FUNCTION_BLOCK FB_BaseMotor

VAR
	mcAxis: 			AXIS_REF;
	eSMState:			E_MoveState;
	
	mcPower: 			MC_Power;
	mcPower_Outputs:	ST_McOutputs;
	
	mcReset: 			MC_Reset;
	mcReset_Outputs:	ST_McOutputs;
	
	mcStop:				MC_Stop;
	mcStop_Outputs:		ST_McOutputs;
	
	mcMoveAbs1: 			MC_MoveAbsolute;
	mcMoveAbs1_Outputs: 	ST_McOutputs;

	mcMoveAbs2: 			MC_MoveAbsolute;
	mcMoveAbs2_Outputs: 	ST_McOutputs;
	
	mcHome:				MC_Home;
	mcHome_Outputs:		ST_McOutputs;
	
END_VAR

(* update the axis status at the beginning of each cycle *)
mcAxis();

(* move axis using a state machine *)
CASE eSMState OF

	MOVESTATE_INIT :	(* initialisation *)
		(* initialize all function blocks *)
		mcMoveAbs1.Execute := FALSE;
		mcReset.Execute := FALSE;
		eSMState := MOVESTATE_ENABLE;

	MOVESTATE_ENABLE :
		mcPower.Enable := TRUE;
		mcPower.Enable_Positive := TRUE;
		mcPower.Enable_Negative := TRUE;
		IF mcPower.Status THEN
			eSMState := MOVESTATE_FORWARD;
		ELSIF mcPower.Error THEN
			eSMState := MOVESTATE_ERROR;
		END_IF

	MOVESTATE_FORWARD :							(* start to first position *)
		mcMoveAbs1.Position := 1500;				(* start to intermediate tartet position *)
		mcMoveAbs1.Velocity := 500;				(* medium velocity level *)
		mcMoveAbs1.BufferMode := MC_Buffered;
		mcMoveAbs1.Execute := TRUE;
		IF mcMoveAbs1.Active  THEN
			(* axis is executing job but is not yet finished *)
			mcMoveAbs1.Execute := FALSE;
			(* leave this state and buffer a second command *)
			eSMState := MOVESTATE_NEWTARGETPOSITION;
		ELSIF mcMoveAbs1.CommandAborted OR mcMoveAbs1.Error THEN
			eSMState := MOVESTATE_ERROR;
		END_IF

	MOVESTATE_NEWTARGETPOSITION :						(* change target position while moving *)
		(* start a buffered motion command while axis is moving *)
		mcMoveAbs2.Position := 5000;						(* start to final target *)
		mcMoveAbs2.Velocity := 1500;						(* increase velocity *)
		mcMoveAbs2.BufferMode := MC_BlendingPrevious; 		(* use velocity of previous command till intermediate target position position *)
		mcMoveAbs2.Execute := TRUE;
		IF mcMoveAbs2.Done THEN
			mcMoveAbs2.Execute := FALSE;
			eSMState := MOVESTATE_BACKWARDS;
		ELSIF mcMoveAbs2.CommandAborted OR mcMoveAbs2.Error THEN
			eSMState := MOVESTATE_ERROR;
		END_IF

	MOVESTATE_BACKWARDS :							(* move back to initial position *)
		mcMoveAbs1.Position := 100;					(* position close to initial position *)
		mcMoveAbs1.Velocity := 2000;				(* high velocity *)
		mcMoveAbs1.BufferMode := MC_Buffered;
		mcMoveAbs1.Execute := TRUE;
		IF mcMoveAbs1.Active THEN
			(* axis is executing job but is not yet finished *)
			mcMoveAbs1.Execute := FALSE;
			(* leave this state and buffer a second command *)
			eSMState := MOVESTATE_BACKWARDSSLOW;
		ELSIF mcMoveAbs1.CommandAborted OR mcMoveAbs1.Error THEN
			eSMState := MOVESTATE_ERROR;
		END_IF

	MOVESTATE_BACKWARDSSLOW :						(* move back to initial position *)
		(* start a buffered motion command while axis is moving *)
		mcMoveAbs2.Position := 0;					(* back to initial position *)
		mcMoveAbs2.Velocity := 100; 				(* slow velocity *)
		mcMoveAbs2.BufferMode := MC_BlendingNext; 	(* use velocity from first target position *)
		mcMoveAbs2.Execute := TRUE;
		IF mcMoveAbs2.Done THEN
			mcMoveAbs2.Execute := FALSE;
			eSMState := MOVESTATE_FORWARD;
		ELSIF mcMoveAbs2.CommandAborted OR mcMoveAbs2.Error THEN
			eSMState := MOVESTATE_ERROR;
		END_IF

	MOVESTATE_ERROR :
		IF mcAxis.Status.Error THEN
			eSMState := MOVESTATE_RESET;			(* axis error requires reset *)
		ELSE
			eSMState := MOVESTATE_INIT;			(* function block errors don't need a reset *)
		END_IF

	MOVESTATE_RESET :
		mcReset.Execute := TRUE;
		IF mcReset.Done THEN
			eSMState := MOVESTATE_INIT;
		ELSIF mcReset.Error THEN
			eSMState := MOVESTATE_INIT; 			(* can't do anything here *)
		END_IF

END_CASE

mcPower(Axis := mcAxis, 
		Enable := mcPower.Enable, 
		Enable_Positive := mcPower.Enable_Positive, 
		Enable_Negative := mcPower.Enable_Negative, 
		Override := 100, 
		Status => mcPower_Outputs.Done, 
		Busy => mcPower_Outputs.Busy, 
		Active => mcPower_Outputs.Active, 
		Error => mcPower_Outputs.Error, 
		ErrorID => mcPower_Outputs.ErrorID);


mcMoveAbs1(Axis := mcAxis,
			Execute := mcMoveAbs1.Execute,
			Position := mcMoveAbs1.Position,
			Velocity := mcMoveAbs1.Velocity,
			BufferMode := mcMoveAbs1.BufferMode,
			Done => mcMoveAbs1_Outputs.Done,
			Busy => mcMoveAbs1_Outputs.Busy,
			Active => mcMoveAbs1_Outputs.Active,
			CommandAborted => mcMoveAbs1_Outputs.CommandAborted,
			Error => mcMoveAbs1_Outputs.Error,
			ErrorID => mcMoveAbs1_Outputs.ErrorID);
			
mcMoveAbs2(Axis := mcAxis,
			Execute := mcMoveAbs1.Execute,
			Position := mcMoveAbs1.Position,
			Velocity := mcMoveAbs1.Velocity,
			BufferMode := mcMoveAbs1.BufferMode,
			Done => mcMoveAbs1_Outputs.Done,
			Busy => mcMoveAbs1_Outputs.Busy,
			Active => mcMoveAbs1_Outputs.Active,
			CommandAborted => mcMoveAbs1_Outputs.CommandAborted,
			Error => mcMoveAbs1_Outputs.Error,
			ErrorID => mcMoveAbs1_Outputs.ErrorID);
			
			
mcReset(Axis := mcAxis,
		Execute := mcReset.Execute,
		Done => mcReset_Outputs.Done,
		Busy => mcReset_Outputs.Busy,
		Error => mcReset_Outputs.Error,
		ErrorID => mcReset_Outputs.ErrorID);
	
// ActPower();	(* call the power function block *)
//ActMove();	(* call the move function block *)
//ActReset();	(* call the reset function block *)

ACTION ActMove:
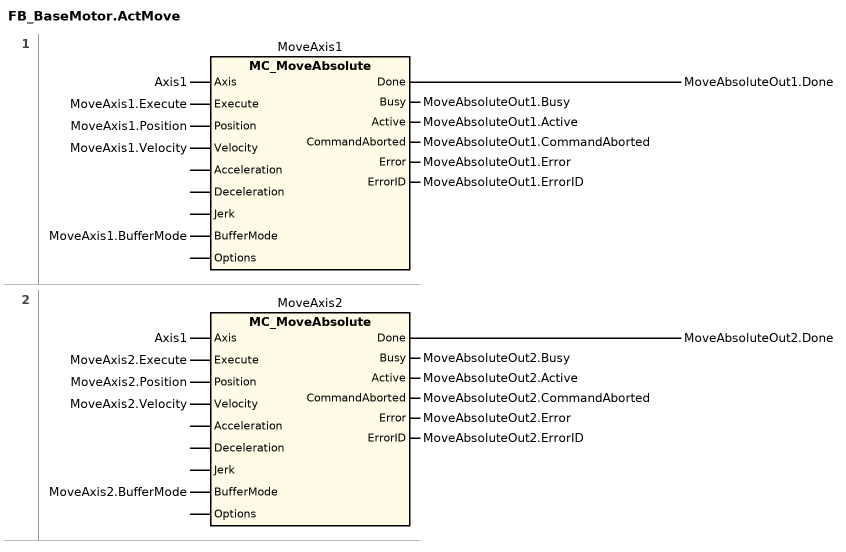
// NETWORK 1
MoveAxis1(
    Axis := Axis1,
    Execute := MoveAxis1.Execute,
    Position := MoveAxis1.Position,
    Velocity := MoveAxis1.Velocity,
    BufferMode := MoveAxis1.BufferMode,
    Busy => MoveAbsoluteOut1.Busy,
    Active => MoveAbsoluteOut1.Active,
    CommandAborted => MoveAbsoluteOut1.CommandAborted,
    Error => MoveAbsoluteOut1.Error,
    ErrorID => MoveAbsoluteOut1.ErrorID); // MC_MoveAbsolute
MoveAbsoluteOut1.Done := MoveAxis1.Done;

// NETWORK 2
MoveAxis2(
    Axis := Axis1,
    Execute := MoveAxis2.Execute,
    Position := MoveAxis2.Position,
    Velocity := MoveAxis2.Velocity,
    BufferMode := MoveAxis2.BufferMode,
    Busy => MoveAbsoluteOut2.Busy,
    Active => MoveAbsoluteOut2.Active,
    CommandAborted => MoveAbsoluteOut2.CommandAborted,
    Error => MoveAbsoluteOut2.Error,
    ErrorID => MoveAbsoluteOut2.ErrorID); // MC_MoveAbsolute
MoveAbsoluteOut2.Done := MoveAxis2.Done;
END_ACTION

ACTION ActPower:
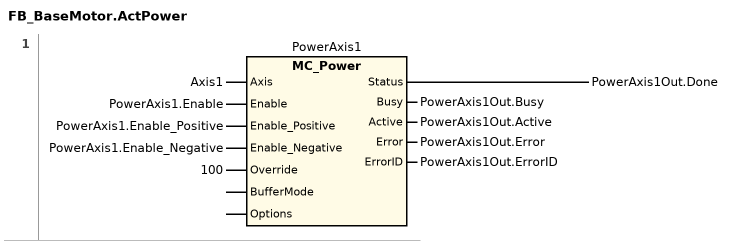
// NETWORK 1
PowerAxis1(
    Axis := Axis1,
    Enable := PowerAxis1.Enable,
    Enable_Positive := PowerAxis1.Enable_Positive,
    Enable_Negative := PowerAxis1.Enable_Negative,
    Override := 100,
    Busy => PowerAxis1Out.Busy,
    Active => PowerAxis1Out.Active,
    Error => PowerAxis1Out.Error,
    ErrorID => PowerAxis1Out.ErrorID); // MC_Power
PowerAxis1Out.Done := PowerAxis1.Status;
END_ACTION

ACTION ActReset:
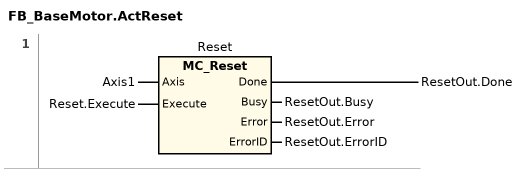
// NETWORK 1
Reset(
    Axis := Axis1,
    Execute := Reset.Execute,
    Busy => ResetOut.Busy,
    Error => ResetOut.Error,
    ErrorID => ResetOut.ErrorID); // MC_Reset
ResetOut.Done := Reset.Done;
END_ACTION

END_FUNCTION_BLOCK

(* stored: Version 1.1.0.1, ProductVersion 3.1.4024.12
   POU FB_BaseMotor: Id {ce2089f9-2565-45a6-999c-d57cf0762d64}, SpecialFunc None
   Action ActMove: Id {3d111008-117e-48c0-b906-ef3dd2ade181}
   Action ActPower: Id {092b2546-15d5-4e2b-a4a8-a0e1930cfd59}
   Action ActReset: Id {6b813b23-b439-4b4e-9388-efe53bb90d5a} *)
